PROGRAM LDDR
VAR
END_VAR

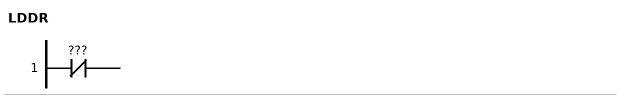
// NETWORK 1

END_PROGRAM

(* stored: Version 1.1.0.1, ProductVersion 3.1.4024.12
   POU LDDR: Id {e6621820-3ff7-4118-bad2-354854e57cd0}, SpecialFunc None *)
